(* CoDeSys 2.3 export: GEN_MODE.EXP *)

(* Data type *)
TYPE GEN_MODE :
	(TRIANGLE:=0,TRIANGLE_POS:=1,SAWTOOTH_RISE:=2,SAWTOOTH_FALL:=3,RECTANGLE:=4,SINUS:=5,COSINUS:=6);
END_TYPE
